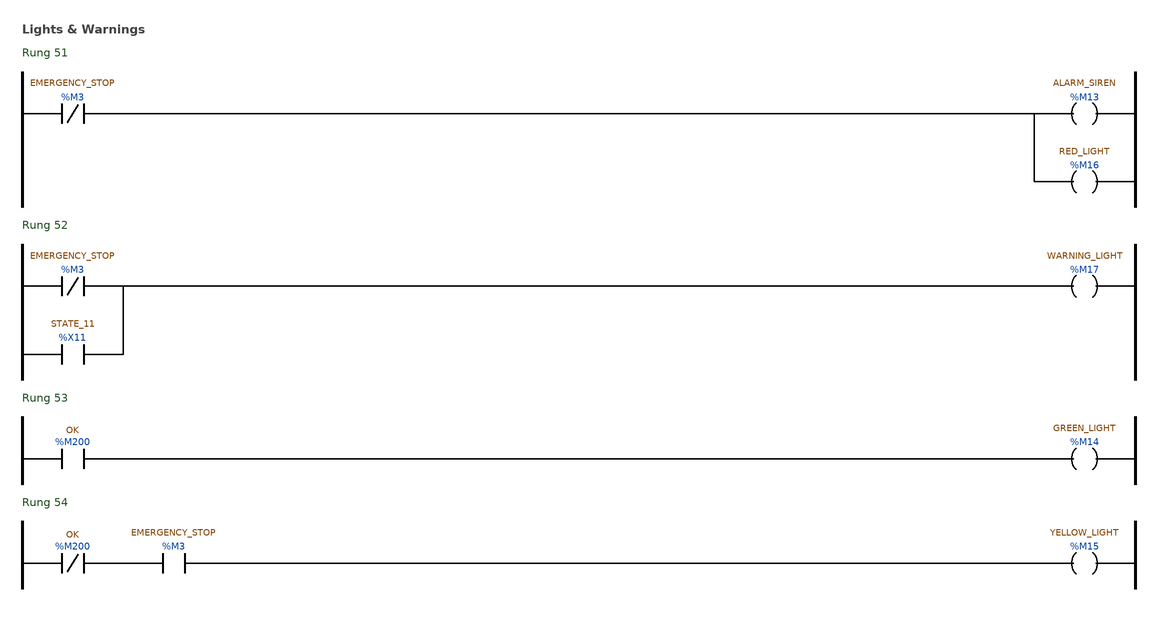
[picture p24: Lights & Warnings, ladder]

// Rung 51
  LDN %M3                 (* EMERGENCY_STOP *)
  ST %M13                 (* ALARM_SIREN *)
  ST %M16                 (* RED_LIGHT *)
  // as ST:
  //   ALARM_SIREN := NOT EMERGENCY_STOP;
  //   RED_LIGHT := NOT EMERGENCY_STOP;

// Rung 52
  LDN %M3                 (* EMERGENCY_STOP *)
  OR %X11                 (* STATE_11 *)
  ST %M17                 (* WARNING_LIGHT *)
  // as ST:
  //   WARNING_LIGHT := NOT EMERGENCY_STOP OR STATE_11;

// Rung 53
  LD %M200                (* OK *)
  ST %M14                 (* GREEN_LIGHT *)
  // as ST:
  //   GREEN_LIGHT := OK;

// Rung 54
  LDN %M200               (* OK *)
  AND %M3                 (* EMERGENCY_STOP *)
  ST %M15                 (* YELLOW_LIGHT *)
  // as ST:
  //   YELLOW_LIGHT := NOT OK AND EMERGENCY_STOP;
